// TIA Portal project "p" (V11)

(* hardware
DEVICE "S7300/ET200 station_1"  SIMATIC 300-Station
   slot 0: "Perfil soporte_0"  Rail  6ES7 390-1***0-0AA0
   slot 2: "PLC_1"  CPU 313C-2 DP  6ES7 313-6CF03-0AB0  V2.6
      slot 0: "Interfaz MPI_1"  MPI
      slot 1: "Interfaz DP_1"  DP
      slot 2: "DI16/DO16_1"  DI16/DO16
      slot 4: "Contaje_1"  Counter
   slot 4: "CP 343-1 Lean_1"  CP 343-1 LEAN  6GK7 343-1CX10-0XE0  V2.4
DEVICE "HMI_1"  KTP600 Basic PN
   slot 0: "HMI"  HMI  6AV6647-0AD11-3AX0  11.0.0
   slot 1: "HMI_RT_1"  KTP600 Basic PN  6AV6647-0AD11-3AX0  11.0.0
   slot 5: "IE_CP_1"  PROFINET interface  IE_CP  V7.1.0
      slot 1: "PROFINET_Interfaz_1"  HMI IE SUBMODULE
         slot 1: "PORT_1"  HMI IE PORTMODULE 1  1.0.0.0
*)

// ===== PLC "PLC_1"  CPU 313C-2 DP =====

VAR_GLOBAL   // PLC tag table "Tabla de variables estándar"
   "UP" AT %M0.0 : Bool;
   "DOWN" AT %M0.1 : Bool;
   "RESET" AT %M0.2 : Bool;
   "PUNTERO" AT %MD10 : DWord;
   "PARALELA" AT %MD14 : DInt;
   "FP1" AT %M50.0 : Bool;
   "FP2" AT %M50.1 : Bool;
   "FP3" AT %M50.2 : Bool;
   "FP4" AT %M50.3 : Bool;
   "FP5" AT %M50.4 : Bool;
   "FP6" AT %M50.5 : Bool;
   "DISPLAY" AT %MB1 : Byte;
   "BIT 0" AT %M1.0 : Bool;
   "BIT 1" AT %M1.1 : Bool;
   "BIT 2" AT %M1.2 : Bool;
   "BIT 3" AT %M1.3 : Bool;
   "BIT 4" AT %M1.4 : Bool;
   "BIT 5" AT %M1.5 : Bool;
   "BIT 6" AT %M1.6 : Bool;
   "P on" AT %M20.0 : Bool;
   "RETURN" AT %M20.1 : Bool;
   "NO_DEC" AT %M20.2 : Bool;
END_VAR

DATA_BLOCK "PUNTEROS"   // DB1
{ S7_Optimized_Access := 'FALSE' }
VERSION : 0.1
   VAR
      DISPLAY : Array [0..9] of Byte;
      "10" : DWord := 10;
   END_VAR
BEGIN
   DISPLAY[0] := B#16#3F;
   DISPLAY[1] := B#16#6;
   DISPLAY[2] := B#16#5B;
   DISPLAY[3] := B#16#4F;
   DISPLAY[4] := B#16#66;
   DISPLAY[5] := B#16#6D;
   DISPLAY[6] := B#16#7D;
   DISPLAY[7] := B#16#7;
   DISPLAY[8] := B#16#7F;
   DISPLAY[9] := B#16#6F;
END_DATA_BLOCK

FUNCTION "Bloque_1" : Void   // FC1, STL
{ S7_Optimized_Access := 'FALSE' }
VERSION : 0.1
   VAR_INPUT
      UP : Bool;
      DOWN : Bool;
      RESET : Bool;
   END_VAR
   VAR_OUTPUT
      DISPALY : Byte;
   END_VAR
BEGIN
END_FUNCTION

ORGANIZATION_BLOCK "Main"   // OB1, STL
TITLE = "Main Program Sweep (Cycle)"
{ S7_Optimized_Access := 'FALSE' }
VERSION : 0.1
   VAR_TEMP
      OB1_EV_CLASS : Byte;   // Bits 0-3 = 1 (Coming event), Bits 4-7 = 1 (Event class 1)
      OB1_SCAN_1 : Byte;   // 1 (Cold restart scan 1 of OB 1), 3 (Scan 2-n of OB 1)
      OB1_PRIORITY : Byte;   // Priority of OB Execution
      OB1_OB_NUMBR : Byte;   // 1 (Organization block 1, OB1)
      OB1_RESERVED_1 : Byte;   // Reserved for system
      OB1_RESERVED_2 : Byte;   // Reserved for system
      OB1_PREV_CYCLE : Int;   // Cycle time of previous OB1 scan (milliseconds)
      OB1_MIN_CYCLE : Int;   // Minimum cycle time of OB1 (milliseconds)
      OB1_MAX_CYCLE : Int;   // Maximum cycle time of OB1 (milliseconds)
      OB1_DATE_TIME : Date_And_Time;   // Date and time OB1 started
   END_VAR
BEGIN

REGION Network 1
         CALL  "Bloque_1"
         ( UP      := "UP",
           DOWN    := "DOWN",
           RESET   := "RESET",
           DISPALY := "DISPLAY"
         );
END_REGION
END_ORGANIZATION_BLOCK

(* ===== HMI "HMI_RT_1" =====
connection "Conexión_HMI": ETHERNET, SIMATIC S7 300/400 MPI

HMI tags "Tabla de variables estándar"
   "RESET" : Bool = PLC "RESET", 1 s
   "DOWN" : Bool = PLC "DOWN", 1 s
   "UP" : Bool = PLC "UP", 1 s
   "BIT 0" : Bool = PLC "BIT 0", 1 s
   "BIT 1" : Bool = PLC "BIT 1", 1 s
   "BIT 2" : Bool = PLC "BIT 2", 1 s
   "BIT 3" : Bool = PLC "BIT 3", 1 s
   "BIT 4" : Bool = PLC "BIT 4", 1 s
   "BIT 5" : Bool = PLC "BIT 5", 1 s
   "BIT 6" : Bool = PLC "BIT 6", 1 s

screen "Imagen_1" 320x240
   Button "Botón_1" at 51,45 size 60x30
   Button "Botón_2" at 51,96 size 60x30
   Button "Botón_3" at 51,149 size 60x30
*)